TYPE ST_BaseTopElement_HMI :
STRUCT
END_STRUCT
END_TYPE

(* stored: Version 1.1.0.1
   DUT ST_BaseTopElement_HMI: Id {b407ef35-511d-0539-2687-37f9a6583220} *)
